{attribute 'qualified_only'}
{attribute 'to_string'}
TYPE E_ModeHandlerStates :
(
	Idle:=0,
	Selftest0,
	Selftest1,
	Selftest2,
	SelftestUndocked,
	Ergonomics1,
	Ergonomics2,
	HaltErgonomics,
	Teleoperation1,
	Teleoperation2,
	EndCase,
	Error
)UINT := Idle
;
END_TYPE

(* stored: Version 1.1.0.1, ProductVersion 3.1.4024.12
   EnumerationTextList E_ModeHandlerStates: Id {976abbab-f0c3-443d-abd1-8326dc118a7e} *)
